Staubli VAL3: buildList.pgx

program buildList()
  local num l_nSize
  local string l_sName
  local num i
  local string l_sMessage
  local tool l_tTool
  local string l_sEmpty
  local string l_sItem
begin
  // INIT the list
  l_sEmpty=""
  call use:stringCopy(l_sEmpty,sList)
  //
  // Build the list
  //
  // get the GUN
  call tcp:getTool(l_tTool,nIndexTool)
  // show the gun
  call tcp:getName(l_sName,nIndexTool)
  call language:message(l_sMessage,21)
  l_sName=l_sMessage+"> "+l_sName
  // create the list
  call listAdd(l_sName)
  l_sItem=("coord  X > "+toString(".2",l_tTool.trsf.x))
  call listAdd(l_sItem)
  l_sItem=("coord  Y > "+toString(".2",l_tTool.trsf.y))
  call listAdd(l_sItem)
  l_sItem=("coord  Z > "+toString(".2",l_tTool.trsf.z))
  call listAdd(l_sItem)
  l_sItem=("coord RX > "+toString(".2",l_tTool.trsf.rx))
  call listAdd(l_sItem)
  l_sItem=("coord RY > "+toString(".2",l_tTool.trsf.ry))
  call listAdd(l_sItem)
  l_sItem=("coord RZ > "+toString(".2",l_tTool.trsf.rz))
  call listAdd(l_sItem)
  // TCP ON OFF
  call language:message(l_sMessage,123)
  call use:strfill(l_sMessage,9,l_sMessage)
  l_sItem=l_sMessage+">ON  "+toString("",l_tTool.otime)+ "mm"
  call listAdd(l_sItem)
  l_sItem=l_sMessage+">OFF "+toString("",l_tTool.ctime)+ "mm"
  call listAdd(l_sItem)
end
